Universal Robots PolyScope program: stacking_p2.urp

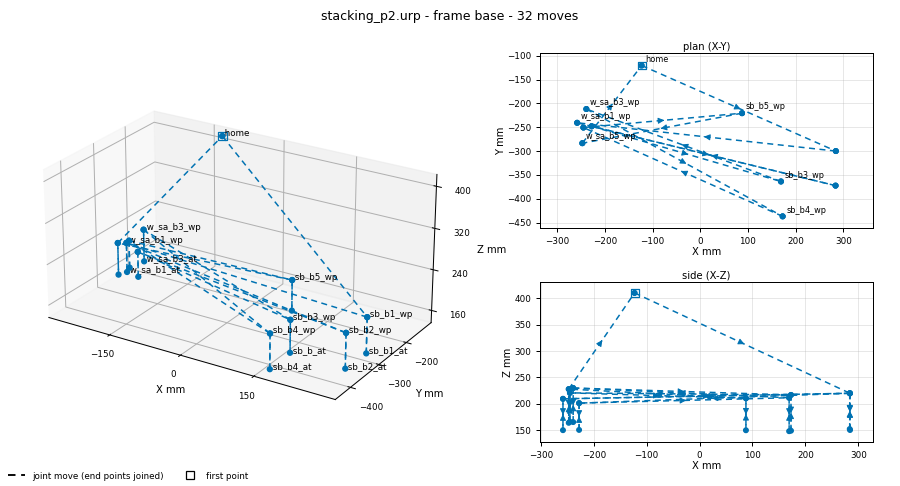
[picture p0: tool path of stacking_p2.urp in frame base, 32 of 32 moves have a stored position in this frame; points joined in program order, loops and branches not executed]
Program stacking_p2 (installation=default directory=/programs/ITER createdIn=5.3.1.64192 lastSavedIn=5.3.1.64192 robotSerialNumber=20195300365)
Calibrated DH parameters: a=[-0.000093, -0.190649, -0.212673, 0.000091, -0.000205, 0]; d=[0.151591, 44.061648, -42.488068, -1.442789, 0.085322, 0.091911]; alpha=[1.570082, -0.003447, 0.007513, 1.572293, -1.571904, 0]; deltaTheta=[0, -0.672656, 0.728185, -0.055522, 0.000005, 0]
Robot Program (runOnlyOnce=true)
  URCap Gripper Activate (Robotiq_Grippers, Robotiq Inc.) dataModel(ResetAndActivateKey=false)
  URCap Gripper (Robotiq_Grippers, Robotiq Inc.) dataModel(position=50.19607843137255, force=100.0, speed=100.0, positionInDouble=50.19607843137255, forceInDouble=100.0, speedInDouble=100.0, slaveIds=[9], blocking=true)
  MoveJ speed 60 deg/s, acceleration 80 deg/s^2 (useActiveTCP=true) feature=Base
    Waypoint home: TCP in base x=-122.938 y=-120.383 z=410.034 mm, rx=2.2731 ry=2.1658 rz=-0.0264 rad; joints [-85.881, -57.164, -80.451, -131.628, 89.647, -263.137] deg
  Folder Stack B
    MoveJ speed 60 deg/s, acceleration 80 deg/s^2 (useActiveTCP=true) feature=Base
      Waypoint sb_b1_wp: TCP in base x=284.372 y=-299.808 z=219.894 mm, rx=2.2369 ry=2.136 rz=0.0122 rad; joints [-28.102, -114.195, -84.199, -68.754, 89.828, -205.167] deg
      Waypoint sb_b1_at: TCP in base x=284.367 y=-299.815 z=150.378 mm, rx=2.2368 ry=2.1359 rz=0.0123 rad; joints [-28.126, -121.493, -93.486, -52.164, 89.765, -205.101] deg; TCP offset x=0 y=0 z=0 mm, rx=0 ry=0 rz=0 rad
      URCap Gripper (Robotiq_Grippers, Robotiq Inc.) dataModel(position=100.0, force=100.0, speed=100.0, positionInDouble=100.0, forceInDouble=100.0, speedInDouble=100.0, slaveIds=[9], blocking=true)
      Waypoint sb_b1_wp: TCP in base x=284.372 y=-299.808 z=219.894 mm, rx=2.2369 ry=2.136 rz=0.0122 rad; joints [-28.102, -114.195, -84.199, -68.754, 89.828, -205.167] deg
      Waypoint w_sa_b1_wp: TCP in base x=-258.271 y=-240.499 z=209.476 mm, rx=3.1151 ry=-0.0825 rz=0.0204 rad; joints [-115.862, -101.636, -103.759, -63.52, 91.564, -202.433] deg
      Waypoint w_sa_b1_at: TCP in base x=-258.276 y=-240.491 z=150.031 mm, rx=3.1151 ry=-0.0827 rz=0.0205 rad; joints [-115.884, -109.689, -111.896, -47.33, 91.487, -202.37] deg
      URCap Gripper (Robotiq_Grippers, Robotiq Inc.) dataModel(position=50.19607843137255, force=100.0, speed=100.0, positionInDouble=50.19607843137255, forceInDouble=100.0, speedInDouble=100.0, slaveIds=[9], blocking=true)
      Waypoint w_sa_b1_wp: TCP in base x=-258.271 y=-240.499 z=209.476 mm, rx=3.1151 ry=-0.0825 rz=0.0204 rad; joints [-115.862, -101.636, -103.759, -63.52, 91.564, -202.433] deg
    MoveJ speed 60 deg/s, acceleration 80 deg/s^2 (useActiveTCP=true) feature=Base
      Waypoint sb_b2_wp: TCP in base x=283.794 y=-372.292 z=220.028 mm, rx=2.2142 ry=2.2013 rz=0.0173 rad; joints [-36.623, -128.603, -60.242, -79.9, 90.737, -216.103] deg
      Waypoint sb_b2_at: TCP in base x=283.771 y=-372.319 z=152.183 mm, rx=2.2142 ry=2.2012 rz=0.0173 rad; joints [-36.654, -133.529, -70.513, -64.699, 90.706, -216.038] deg
      URCap Gripper (Robotiq_Grippers, Robotiq Inc.) dataModel(position=100.0, force=100.0, speed=100.0, positionInDouble=100.0, forceInDouble=100.0, speedInDouble=100.0, slaveIds=[9], blocking=true)
      Waypoint sb_b2_wp: TCP in base x=283.794 y=-372.292 z=220.028 mm, rx=2.2142 ry=2.2013 rz=0.0173 rad; joints [-36.623, -128.603, -60.242, -79.9, 90.737, -216.103] deg
      Waypoint w_sa_b2_wp: TCP in base x=-227.79 y=-247.903 z=201.3 mm, rx=-3.1116 ry=0.1046 rz=-0.0512 rad; joints [-110.33, -99.289, -107.723, -65.024, 91.583, -196.119] deg
      Waypoint w_sa_b2_at: TCP in base x=-227.812 y=-247.879 z=150.535 mm, rx=-3.1115 ry=0.1048 rz=-0.0512 rad; joints [-110.354, -106.436, -114.862, -50.742, 91.515, -196.061] deg
      URCap Gripper (Robotiq_Grippers, Robotiq Inc.) dataModel(position=50.19607843137255, force=100.0, speed=100.0, positionInDouble=50.19607843137255, forceInDouble=100.0, speedInDouble=100.0, slaveIds=[9], blocking=true)
      Waypoint w_sa_b2_wp: TCP in base x=-227.79 y=-247.903 z=201.3 mm, rx=-3.1116 ry=0.1046 rz=-0.0512 rad; joints [-110.33, -99.289, -107.723, -65.024, 91.583, -196.119] deg
    MoveJ speed 60 deg/s, acceleration 80 deg/s^2 (useActiveTCP=true) feature=Base
      Waypoint sb_b3_wp: TCP in base x=169.247 y=-363.593 z=211.49 mm, rx=2.1909 ry=2.2024 rz=0.0037 rad; joints [-46.21, -112.261, -89.113, -66.558, 90.453, -226.181] deg
      Waypoint sb_b_at: TCP in base x=169.246 y=-363.592 z=148.111 mm, rx=2.1909 ry=2.2024 rz=0.0037 rad; joints [-46.23, -119.472, -97.295, -51.168, 90.39, -226.121] deg; TCP offset x=0 y=0 z=0 mm, rx=0 ry=0 rz=0 rad
      URCap Gripper (Robotiq_Grippers, Robotiq Inc.) dataModel(position=100.0, force=100.0, speed=100.0, positionInDouble=100.0, forceInDouble=100.0, speedInDouble=100.0, slaveIds=[9], blocking=true)
      Waypoint sb_b3_wp: TCP in base x=169.247 y=-363.593 z=211.49 mm, rx=2.1909 ry=2.2024 rz=0.0037 rad; joints [-46.21, -112.261, -89.113, -66.558, 90.453, -226.181] deg
      Waypoint w_sa_b3_wp: TCP in base x=-238.98 y=-211.657 z=229.948 mm, rx=-2.2294 ry=-2.1838 rz=0.0163 rad; joints [-114.112, -91.23, -109.254, -69.34, 88.995, -292.564] deg
      Waypoint w_sa_b3_at: TCP in base x=-238.979 y=-211.665 z=165.424 mm, rx=-2.2294 ry=-2.1838 rz=0.0165 rad; joints [-114.14, -99.517, -120.015, -50.29, 88.908, -292.484] deg
      URCap Gripper (Robotiq_Grippers, Robotiq Inc.) dataModel(position=50.19607843137255, force=100.0, speed=100.0, positionInDouble=50.19607843137255, forceInDouble=100.0, speedInDouble=100.0, slaveIds=[9], blocking=true)
      Waypoint w_sa_b3_wp: TCP in base x=-238.98 y=-211.657 z=229.948 mm, rx=-2.2294 ry=-2.1838 rz=0.0163 rad; joints [-114.112, -91.23, -109.254, -69.34, 88.995, -292.564] deg
    MoveJ speed 60 deg/s, acceleration 80 deg/s^2 (useActiveTCP=true) feature=Base
      Waypoint sb_b4_wp: TCP in base x=172.769 y=-436.751 z=216.834 mm, rx=2.2461 ry=2.1748 rz=-0.0044 rad; joints [-52.304, -129.217, -59.921, -79.919, 90.209, -230.281] deg
      Waypoint sb_b4_at: TCP in base x=172.746 y=-436.763 z=149.006 mm, rx=2.2461 ry=2.1748 rz=-0.0044 rad; joints [-52.333, -134.228, -69.998, -64.832, 90.179, -230.215] deg; TCP offset x=0 y=0 z=0 mm, rx=0 ry=0 rz=0 rad
      URCap Gripper (Robotiq_Grippers, Robotiq Inc.) dataModel(position=100.0, force=100.0, speed=100.0, positionInDouble=100.0, forceInDouble=100.0, speedInDouble=100.0, slaveIds=[9], blocking=true)
      Waypoint sb_b4_wp: TCP in base x=172.769 y=-436.751 z=216.834 mm, rx=2.2461 ry=2.1748 rz=-0.0044 rad; joints [-52.304, -129.217, -59.921, -79.919, 90.209, -230.281] deg
      Waypoint w_sa_b4_wp: TCP in base x=-245.189 y=-250.465 z=220.693 mm, rx=2.2499 ry=2.1886 rz=-0.0042 rad; joints [-112.717, -99.979, -102.147, -67.604, 90.389, -290.778] deg
      Waypoint w_sa_b4_at: TCP in base x=-245.197 y=-250.444 z=165.926 mm, rx=2.25 ry=2.1885 rz=-0.0041 rad; joints [-112.742, -106.561, -110.516, -52.658, 90.325, -290.716] deg
      URCap Gripper (Robotiq_Grippers, Robotiq Inc.) dataModel(position=50.19607843137255, force=100.0, speed=100.0, positionInDouble=50.19607843137255, forceInDouble=100.0, speedInDouble=100.0, slaveIds=[9], blocking=true)
      Waypoint w_sa_b4_wp: TCP in base x=-245.189 y=-250.465 z=220.693 mm, rx=2.2499 ry=2.1886 rz=-0.0042 rad; joints [-112.717, -99.979, -102.147, -67.604, 90.389, -290.778] deg
    MoveJ speed 60 deg/s, acceleration 80 deg/s^2 (useActiveTCP=true) feature=Base
      Waypoint sb_b5_wp: TCP in base x=87.61 y=-220.378 z=210.477 mm, rx=2.2119 ry=2.1926 rz=0.0266 rad; joints [-35.573, -69.277, -133.023, -65.94, 91.083, -214.634] deg
      Waypoint sb_b5_at: TCP in base x=87.587 y=-220.373 z=149.892 mm, rx=2.212 ry=2.1925 rz=0.0266 rad; joints [-35.613, -81.407, -144.951, -41.885, 90.95, -214.536] deg; TCP offset x=0 y=0 z=0 mm, rx=0 ry=0 rz=0 rad
      URCap Gripper (Robotiq_Grippers, Robotiq Inc.) dataModel(position=100.0, force=100.0, speed=100.0, positionInDouble=100.0, forceInDouble=100.0, speedInDouble=100.0, slaveIds=[9], blocking=true)
      Waypoint sb_b5_wp: TCP in base x=87.61 y=-220.378 z=210.477 mm, rx=2.2119 ry=2.1926 rz=0.0266 rad; joints [-35.573, -69.277, -133.023, -65.94, 91.083, -214.634] deg
      Waypoint w_sa_b5_wp: TCP in base x=-247.393 y=-283.334 z=227.844 mm, rx=2.2495 ry=2.1402 rz=-0.0127 rad; joints [-111.4, -105.454, -93.637, -69.526, 91.99, -288.199] deg
      Waypoint w_sa_b5_at: TCP in base x=-247.399 y=-283.319 z=164.004 mm, rx=2.2496 ry=2.1402 rz=-0.0126 rad; joints [-111.426, -112.371, -103.175, -53.072, 91.924, -288.131] deg
      URCap Gripper (Robotiq_Grippers, Robotiq Inc.) dataModel(position=50.19607843137255, force=100.0, speed=100.0, positionInDouble=50.19607843137255, forceInDouble=100.0, speedInDouble=100.0, slaveIds=[9], blocking=true)
      Waypoint w_sa_b5_wp: TCP in base x=-247.393 y=-283.334 z=227.844 mm, rx=2.2495 ry=2.1402 rz=-0.0127 rad; joints [-111.4, -105.454, -93.637, -69.526, 91.99, -288.199] deg
  MoveJ speed 60 deg/s, acceleration 80 deg/s^2 (useActiveTCP=true) feature=Base
    Waypoint home: TCP in base x=-122.938 y=-120.383 z=410.034 mm, rx=2.2731 ry=2.1658 rz=-0.0264 rad; joints [-85.881, -57.164, -80.451, -131.628, 89.647, -263.137] deg
